INTERFACE I_Initializable EXTENDS I_Base

METHOD Initialize
END_METHOD

{attribute 'monitoring' := 'call'}
PROPERTY Initialized : BOOL
GET
END_GET
SET
END_SET
END_PROPERTY

END_INTERFACE

(* stored: Version 1.1.0.1, ProductVersion 3.1.4026.18
   Itf I_Initializable: Id {aaea7e7e-41a5-49c1-8b5d-cd842bb624f2}
   Method Initialize: Id {c9c29a0b-548d-4d02-8fcc-ef709b07aa61}
   Property Initialized: Id {dc50bae1-6ce1-45d0-9786-31d4c490340a}
   Get Get: Id {c0c3f9e9-cc4d-4aa4-965e-533aeb972726}
   Set Set: Id {2368bccd-c88d-40f4-a277-c70194ded820} *)
